TYPE ST_Tank :
STRUCT
	
	id : INT;
	temperature : REAL;
    level : REAL;
	alarm : BOOL ;
	
END_STRUCT
END_TYPE

(* stored: Version 1.1.0.1, ProductVersion 3.1.4024.16
   DUT ST_Tank: Id {48be6a43-a4e5-4e91-876b-572157165462} *)
